Universal Robots PolyScope program: event_115.urp

Program event_115 (createdIn=3.2.19293 lastSavedIn=3.2.19293 directory=/programs installation=default robotSerialNumber=2015351391)
Calibrated DH parameters: a=[0.000352, -0.161198, -0.373486, 0.00005, 0.000049, 0]; d=[0.089268, 352.477598, -320.08558, -32.281492, 0.094939, 0.082518]; alpha=[1.570728, 0.001116, -0.003686, 1.571189, -1.570572, 0]; deltaTheta=[-0.000012, 1.181849, -1.491165, 0.309495, -0.000007, 0.000025]
Robot Program (runOnlyOnce=false motionType=MoveJ speed=1.047198 acceleration=1.396263 recalculateMotions=false)
  MoveL speed 250 mm/s, acceleration 1200 mm/s^2 (recalculateMotions=false) feature=Base
    Waypoint waypoint1: TCP in base x=239.013 y=198.822 z=690.646 mm, rx=-1.5849 ry=-0.1112 rz=-0.2807 rad; joints [52.537, -69.916, -94.003, -17.001, 121.19, -14.989] deg
    Waypoint waypoint2: TCP in base x=239.013 y=198.808 z=490.015 mm, rx=-1.5849 ry=-0.1114 rz=-0.2807 rad; joints [52.474, -69.278, -124.059, 12.438, 121.352, -14.959] deg
Event  expression=Button≟ True
  Halt
